{attribute 'qualified_only'}
VAR_GLOBAL
	// DALI 2
	kl6821_01_rpcResp 			: ST_DALIBridgeResponse;
	kl6821_01_notif				: ST_DALIBridgeNotification;
	kl6821_01_bridge			: FB_DALIBridge(Communication.aKL6821Communication[1]);
END_VAR

(* stored: Version 1.1.0.1, ProductVersion 3.1.4024.11
   GVL GVL_DALI_Bus: Id {98babae1-1edc-4d37-95bb-a0c997317828} *)
